FUNCTION_BLOCK FB_MotorAbb880_malli IMPLEMENTS I_Motor

VAR CONSTANT
	cScale				: REAL := 200.0;	// 1 % = 200 (100 % = 20000, vrt. ACS880 par. 46.01)
	cStopSpeedLimit		: REAL := 2.0;		// [%] tämän alle -> ajo voidaan estää pysäytyksessä
END_VAR

VAR
	// --- Prosessikuva
	stControlWord		AT %Q* : ST_ControlWord;
	stStatusWord		AT %I* : ST_StatusWord;
	nSpeedRef			AT %Q* : INT;
	nSpeedActual		AT %I* : INT;

	_bInit				: BOOL;
	_refHmi				: REFERENCE TO ST_Motors;

	// --- Komennot (propertyjen kautta)
	_bEnable			: BOOL;			// Taajuusmuuttajan päävirta/valmius (SwitchOn)
	_bAuto				: BOOL;			// Käyntikäsky automaattiajossa
	_nSpeed				: INT;			// Nopeusohje automaattiajossa [%]
	_bManual			: BOOL;			// Valinta: TRUE = käsiajo, FALSE = automaatti
	_bManualFwd			: BOOL;			// Käsiajo eteen (pidä painettuna)
	_bManualRev			: BOOL;			// Käsiajo taakse (pidä painettuna)
	_fManualSpeed		: REAL := 10.0;	// Käsiajon nopeus [%]
	_fManualMax			: REAL := 20.0;	// Käsiajon nopeusraja [%]
	_bReset				: BOOL;			// Vikakuittaus
	_bQuickStop			: BOOL;			// TRUE = pikapysäytys (kytke NC-hätäseisoista: NOT bOk)

	// --- Sisäiset
	_eState				: (DRV_DISABLED := 0, DRV_READY, DRV_SWITCHED_ON, DRV_RUNNING, DRV_FAULT);
	_bActiveManual		: BOOL;			// Oikeasti käytössä oleva ajotapa
	_bRunInhibit		: BOOL;			// Vaatii uuden käynnistyskäskyn (tilanvaihto/vian jälkeen)
	_bPowerReq			: BOOL;
	_bRunReq			: BOOL;
	_fSpeedCmd			: REAL;
	_fSpeedRef			: REAL;
	_fSpeedActual		: REAL;
	_tStopTimeout		: TIME := T#10S;	// Max aika hallittuun pysäytykseen

	bRunRaw				: BOOL;
	bModeChangePending	: BOOL;
	bStopping			: BOOL;
	bKeepOperation		: BOOL;
	bWaiting			: BOOL;

	_rtReset			: R_TRIG;
	_tpReset			: TP;
	_tonStop			: TON;
	_tonWatch			: TON;
END_VAR

HmiCommands();

// ============================================================
// 1. Tilan tulkinta statussanasta (CiA 402 -tilakone)
// ============================================================
IF stStatusWord.Fault THEN
    _eState := DRV_FAULT;
ELSIF stStatusWord.OperationEnabled THEN
    _eState := DRV_RUNNING;
ELSIF stStatusWord.SwitchedOn THEN
    _eState := DRV_SWITCHED_ON;
ELSIF stStatusWord.ReadyToSwitchOn THEN
    _eState := DRV_READY;
ELSE
    _eState := DRV_DISABLED;     // Not ready / Switch on disabled
END_IF

_fSpeedActual := INT_TO_REAL(nSpeedActual) / cScale;

// ============================================================
// 2. Ajotavan valinta (vaihto vain pysäytettynä)
// ============================================================
bModeChangePending := (_bManual <> _bActiveManual);
IF bModeChangePending AND (_eState <> DRV_RUNNING) THEN
    _bActiveManual     := _bManual;
    _bRunInhibit       := TRUE;          // ei automaattista käynnistystä vaihdon jälkeen
    bModeChangePending := FALSE;
END_IF

IF _bActiveManual THEN
    bRunRaw    := _bManualFwd XOR _bManualRev;
    _fSpeedCmd := LIMIT(0.0, _fManualSpeed, _fManualMax);
    IF _bManualRev THEN
        _fSpeedCmd := -_fSpeedCmd;
    END_IF
ELSE
    bRunRaw    := _bAuto;
    _fSpeedCmd := LIMIT(-100.0, INT_TO_REAL(_nSpeed), 100.0);   // rajaa 0..100 jos peruutus ei sallittu
END_IF

IF bModeChangePending THEN
    bRunRaw := FALSE;                    // pysäytä ensin
END_IF

// ============================================================
// 3. Käyntiluvat
// ============================================================
IF _eState = DRV_FAULT THEN
    _bRunInhibit := TRUE;                // vian jälkeen vaaditaan uusi käynnistyskäsky
END_IF
IF NOT bRunRaw THEN
    _bRunInhibit := FALSE;
END_IF

_bPowerReq := _bEnable AND NOT _bQuickStop;
_bRunReq   := _bPowerReq AND bRunRaw AND NOT _bRunInhibit;

// Hallittu pysäytys: nopeusohje 0 -> odota kunnes pysähtynyt (tai timeout) -> EnableOperation pois
bStopping      := (_eState = DRV_RUNNING) AND NOT _bRunReq AND _bPowerReq;
_tonStop(IN := bStopping, PT := _tStopTimeout);
bKeepOperation := bStopping AND (ABS(_fSpeedActual) > cStopSpeedLimit) AND NOT _tonStop.Q;

// Valvonta: pyydetty tila ei toteudu 5 s kuluessa (STO, local-tila, kenttäväylä...)
bWaiting := (_bPowerReq AND (_eState = DRV_DISABLED OR _eState = DRV_READY))
         OR (_bRunReq   AND _eState = DRV_SWITCHED_ON);
_tonWatch(IN := bWaiting, PT := T#5S);

// ============================================================
// 4. Vikakuittaus — nouseva reuna, pulssi 200 ms
// ============================================================
_rtReset(CLK := _bReset);
_tpReset(IN := _rtReset.Q AND (_eState = DRV_FAULT), PT := T#200MS);
stControlWord.FaultReset := _tpReset.Q;

// ============================================================
// 5. Ohjaussana
// ============================================================
IF _eState = DRV_FAULT THEN
    // Vika: disable voltage, odotetaan kuittausta
    stControlWord.SwitchOn        := FALSE;
    stControlWord.EnableVoltage   := FALSE;
    stControlWord.QuickStop       := TRUE;
    stControlWord.EnableOperation := FALSE;

ELSIF _bQuickStop THEN
    // Quick stop
    stControlWord.SwitchOn        := FALSE;
    stControlWord.EnableVoltage   := TRUE;
    stControlWord.QuickStop       := FALSE;
    stControlWord.EnableOperation := FALSE;

ELSIF NOT _bEnable THEN
    // Shutdown
    stControlWord.SwitchOn        := FALSE;
    stControlWord.EnableVoltage   := TRUE;
    stControlWord.QuickStop       := TRUE;
    stControlWord.EnableOperation := FALSE;

ELSE
    stControlWord.EnableVoltage   := TRUE;
    stControlWord.QuickStop       := TRUE;
    CASE _eState OF
        DRV_DISABLED:       // Shutdown
            stControlWord.SwitchOn        := FALSE;
            stControlWord.EnableOperation := FALSE;
        DRV_READY:          // Switch on
            stControlWord.SwitchOn        := TRUE;
            stControlWord.EnableOperation := FALSE;
        DRV_SWITCHED_ON:    // Enable operation vain käyntikäskyllä
            stControlWord.SwitchOn        := TRUE;
            stControlWord.EnableOperation := _bRunReq;
        DRV_RUNNING:
            stControlWord.SwitchOn        := TRUE;
            stControlWord.EnableOperation := _bRunReq OR bKeepOperation;
    END_CASE
END_IF

// ============================================================
// 6. Nopeusohje (-100..100 % -> -20000..20000)
// ============================================================
IF _bRunReq THEN
    _fSpeedRef := _fSpeedCmd;
ELSE
    _fSpeedRef := 0.0;                   // pysäytys ramppia pitkin ajon aikana
END_IF
nSpeedRef := REAL_TO_INT(LIMIT(-100.0, _fSpeedRef, 100.0) * cScale);

PROPERTY bAuto : BOOL
GET
bAuto := _bAuto;
END_GET
SET
_bAuto := bAuto;
END_SET
END_PROPERTY

PROPERTY bEnable : BOOL
GET
bEnable := _bEnable;
END_GET
SET
_bEnable := bEnable;
END_SET
END_PROPERTY

PROPERTY bFault : BOOL
GET
bFault := _eState = DRV_FAULT;
END_GET
END_PROPERTY

PROPERTY bManual : BOOL
GET
bManual := _bManual;
END_GET
SET
_bManual := bManual;
END_SET
END_PROPERTY

PROPERTY bManualActive : BOOL
GET
bManualActive := _bActiveManual;
END_GET
END_PROPERTY

PROPERTY bManualFwd : BOOL
SET
_bManualFwd := bManualFwd;
END_SET
END_PROPERTY

PROPERTY bManualRev : BOOL
SET
_bManualRev := bManualRev;
END_SET
END_PROPERTY

PROPERTY bQuickStop : BOOL
SET
_bQuickStop := bQuickStop OR _refHmi.bStop;
END_SET
END_PROPERTY

PROPERTY bReset : BOOL
SET
_bReset := bReset;
END_SET
END_PROPERTY

PROPERTY bRunning : BOOL
GET
bRunning := _eState = DRV_RUNNING;
END_GET
END_PROPERTY

PROPERTY bTimeout : BOOL
GET
bTimeout := _tonWatch.Q;
END_GET
END_PROPERTY

//FB_Init is always available implicitly and it is used primarily for initialization.
//The return value is not evaluated. For a specific influence, you can also declare the
//methods explicitly and provide additional code there with the standard initialization
//code. You can evaluate the return value.
METHOD FB_Init: BOOL
VAR_INPUT
    bInitRetains: BOOL; // TRUE: the retain variables are initialized (reset warm / reset cold)
    bInCopyCode: BOOL;  // TRUE: the instance will be copied to the copy code afterward (online change)   
END_VAR
_bInit := TRUE;
END_METHOD

PROPERTY fManualSpeed : REAL
GET
fManualSpeed := _fManualSpeed;
END_GET
SET
 IF _refHmi.nManualSpeed > fManualSpeed THEN
	_fManualSpeed := _refHmi.nManualSpeed;
ELSE
	_fManualSpeed := fManualSpeed;
END_IF
END_SET
END_PROPERTY

PROPERTY fSpeedActual : REAL
GET
fSpeedActual := _fSpeedActual;
END_GET
END_PROPERTY

METHOD INTERNAL HmiCommands
VAR_INPUT
END_VAR
bAuto := _refHmi.bAuto;
bManual := _refHmi.bManual AND NOT _refHmi.bAuto;
END_METHOD

METHOD Init
VAR_INPUT
	sName		: STRING;
	refHmi		: REFERENCE TO ST_Motors;
END_VAR
IF _binit THEN
	_refHmi REF= refHmi;
	_refHmi.sName := sName;
END_IF
END_METHOD

PROPERTY nSpeed : INT
GET
nSpeed := _nSpeed;
END_GET
SET
_nSpeed := nSpeed;
END_SET
END_PROPERTY

PROPERTY nState : INT
GET
nState := TO_INT(_eState);
END_GET
END_PROPERTY

END_FUNCTION_BLOCK

(* stored: Version 1.1.0.1
   POU FB_MotorAbb880_malli: Id {eafde16a-d9d2-49c8-9aef-75aff923c034}, SpecialFunc None
   Property bAuto: Id {8618881a-181e-4799-b984-84ef869dd1bb}
   Get Get: Id {d9d98bf6-fec5-4a69-946e-fc62f09273af}
   Set Set: Id {e362960b-616c-4838-a45f-4b90912d678c}
   Property bEnable: Id {8f9a9245-ec9e-43b7-80e3-36e7354c902d}
   Get Get: Id {afe158e3-af94-493a-9b93-41db75825348}
   Set Set: Id {de86dc6e-e117-4807-bf7f-e1a8335cec0f}
   Property bFault: Id {d2c2bee8-03ea-4580-a1b1-62e31918905a}
   Get Get: Id {1545711b-157f-4413-838f-470acb7dd06e}
   Property bManual: Id {a2d4a816-621c-4707-abc5-6754bb84ee44}
   Get Get: Id {028e3361-eccb-48e6-9952-f0c7e8e93cef}
   Set Set: Id {f459f5de-44ec-4620-b5e3-e8863197d107}
   Property bManualActive: Id {11b8a966-ddcf-4050-9056-f4c6f83eeb5a}
   Get Get: Id {cde5e8a9-62e1-484a-b2c5-9653bf71a0a2}
   Property bManualFwd: Id {552f7125-b6eb-47ba-a36d-397fc7f6607a}
   Set Set: Id {e7e1c9d3-6c41-430b-977c-2b43cbbeddc9}
   Property bManualRev: Id {1e6c91ed-1039-42a1-aee3-c9fe29a86b00}
   Set Set: Id {22481690-3ddd-493d-84f5-bb7f4a3e2133}
   Property bQuickStop: Id {3120ea7f-5688-4b97-a306-b8e2924a4092}
   Set Set: Id {0fe082d1-d38c-4766-b80b-fc61c6565aa9}
   Property bReset: Id {16a94efa-b997-4702-86eb-e98c13bfc6f9}
   Set Set: Id {48db6ad1-de65-495d-8e42-e033417b982a}
   Property bRunning: Id {1fa4d785-3f7a-4693-a48d-02d477c4a06b}
   Get Get: Id {a2c81aef-a803-4d32-b331-218a0f0deecf}
   Property bTimeout: Id {93301c03-51b7-4812-9e5e-411ff6799f02}
   Get Get: Id {43a02fc7-62b2-41cc-ad48-f80838c9c016}
   Method FB_Init: Id {fcd88a25-239f-459f-b4dc-8b11ef31c357}
   Property fManualSpeed: Id {201eb5e4-613a-49ed-9556-d99a3d7f46c7}
   Get Get: Id {710872eb-27b5-4a66-8189-6702bd092504}
   Set Set: Id {63658fb3-e55f-4156-89fc-474ba76971a6}
   Property fSpeedActual: Id {74a36abc-7604-4a50-99a2-c697211935ef}
   Get Get: Id {5a3feee0-bada-41c8-9032-0ce61cb2087f}
   Method HmiCommands: Id {4c850631-6bc7-4e13-9386-e1642356329b}
   Method Init: Id {d510b2bb-44fc-4979-8d98-a0c064f5975d}
   Property nSpeed: Id {20836442-a0ca-4dab-9f25-5119f1241edc}
   Get Get: Id {5f74a9b1-97e6-463c-8416-264b79875f41}
   Set Set: Id {e2ffacf8-c223-4b56-adc6-aa640c09c76e}
   Property nState: Id {efcede8a-cb95-49cc-b265-4dcad6a08c83}
   Get Get: Id {cbb649ab-360d-4341-8c17-ce7f43e50183} *)
